TYPE UDT_Estop_RD :
STRUCT
input        : BOOL;
notEstop     : BOOL;
disable      : BOOL;
END_STRUCT
END_TYPE

(* stored: Version 1.1.0.1, ProductVersion 3.1.4024.12
   DUT UDT_Estop_RD: Id {3017cc5c-7a8c-4561-b9b6-2fe1cc46e40a} *)
